% RSLogix 500 project DIGITAL_CONTROL_LOGIC_BAK014.RSS, saved by version 12.00.00.00 %
PROJECT "DRACOFS"    % processor: Bul.1763 MicroLogix 1100 Series B %

PROGRAM FILES
  LAD 2 "MAIN"  3 rungs
  LAD 4 "DIGITAL IO"  5 rungs
  LAD 5 "CONTROL"  10 rungs

DATA FILES
  O0 OUTPUT  5 elements
  I1 INPUT  7 elements
  S2 STATUS  66 elements
  B3 BINARY  1 elements
  T4 TIMER  3 elements
  C5 COUNTER  1 elements
  R6 CONTROL  1 elements
  N7 INTEGER  1 elements
  F8 FLOAT  1 elements

LADDER 2 "MAIN"
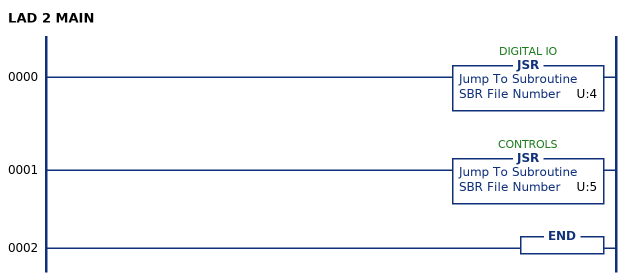
% Rung: 0 %
SOR JSR U:4 EOR
%   U:4  "DIGITAL IO" %
% Rung: 1 %
SOR JSR U:5 EOR
%   U:5  "CONTROLS" %
% Rung: 2 %
SOR END EOR

LADDER 4 "DIGITAL IO"
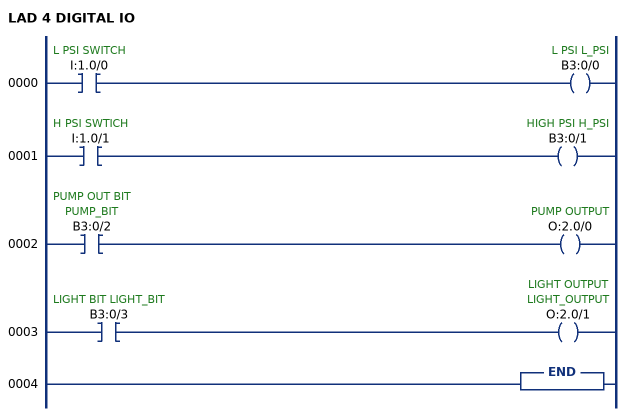
% Rung: 0 %
SOR XIC I:1.0/0 OTE B3:0/0 EOR
%   I:1.0/0  "L PSI SWITCH" %
%   B3:0/0  L_PSI  "L PSI" %
% Rung: 1 %
SOR XIC I:1.0/1 OTE B3:0/1 EOR
%   I:1.0/1  "H PSI SWTICH" %
%   B3:0/1  H_PSI  "HIGH PSI" %
% Rung: 2 %
SOR XIC B3:0/2 OTE O:2.0/0 EOR
%   B3:0/2  PUMP_BIT  "PUMP OUT BIT" %
%   O:2.0/0  "PUMP OUTPUT" %
% Rung: 3 %
SOR XIC B3:0/3 OTE O:2.0/1 EOR
%   B3:0/3  LIGHT_BIT  "LIGHT BIT" %
%   O:2.0/1  LIGHT_OUTPUT  "LIGHT OUTPUT" %
% Rung: 4 %
SOR END EOR

LADDER 5 "CONTROL"
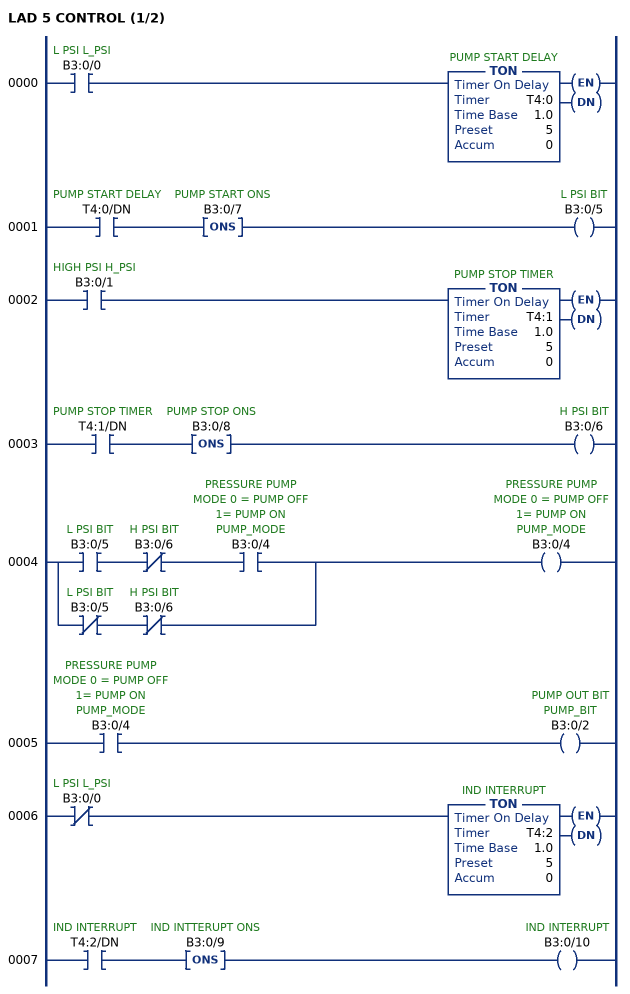
% Rung: 0 %
SOR XIC B3:0/0 TON T4:0 1.0 5 0 EOR
%   B3:0/0  L_PSI  "L PSI" %
%   T4:0  "PUMP START DELAY" %
% Rung: 1 %
SOR XIC T4:0/DN ONS B3:0/7 OTE B3:0/5 EOR
%   T4:0  "PUMP START DELAY" %
%   B3:0/7  "PUMP START ONS" %
%   B3:0/5  "L PSI BIT" %
% Rung: 2 %
SOR XIC B3:0/1 TON T4:1 1.0 5 0 EOR
%   B3:0/1  H_PSI  "HIGH PSI" %
%   T4:1  "PUMP STOP TIMER" %
% Rung: 3 %
SOR XIC T4:1/DN ONS B3:0/8 OTE B3:0/6 EOR
%   T4:1  "PUMP STOP TIMER" %
%   B3:0/8  "PUMP STOP ONS" %
%   B3:0/6  "H PSI BIT" %
% Rung: 4 %
SOR BST XIC B3:0/5 XIO B3:0/6 XIC B3:0/4 NXB XIO B3:0/5 XIO B3:0/6 BND OTE B3:0/4 EOR
%   B3:0/5  "L PSI BIT" %
%   B3:0/6  "H PSI BIT" %
%   B3:0/4  PUMP_MODE  "PRESSURE PUMP MODE 0 = PUMP OFF 1= PUMP ON" %
% Rung: 5 %
SOR XIC B3:0/4 OTE B3:0/2 EOR
%   B3:0/4  PUMP_MODE  "PRESSURE PUMP MODE 0 = PUMP OFF 1= PUMP ON" %
%   B3:0/2  PUMP_BIT  "PUMP OUT BIT" %
% Rung: 6 %
SOR XIO B3:0/0 TON T4:2 1.0 5 0 EOR
%   B3:0/0  L_PSI  "L PSI" %
%   T4:2  "IND INTERRUPT" %
% Rung: 7 %
SOR XIC T4:2/DN ONS B3:0/9 OTE B3:0/10 EOR
%   T4:2  "IND INTERRUPT" %
%   B3:0/9  "IND INTTERUPT ONS" %
%   B3:0/10  "IND INTERRUPT" %

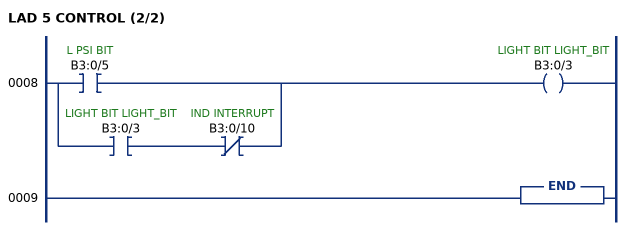
% Rung: 8 %
SOR BST XIC B3:0/5 NXB XIC B3:0/3 XIO B3:0/10 BND OTE B3:0/3 EOR
%   B3:0/5  "L PSI BIT" %
%   B3:0/3  LIGHT_BIT  "LIGHT BIT" %
%   B3:0/10  "IND INTERRUPT" %
% Rung: 9 %
SOR END EOR

DATA TABLE (non-zero values as saved)
DATA B3
% B3:0 % 0X0068
DATA T4
% .PRE .ACC %
% T4:0 % 5 0
% T4:1 % 5 0
% T4:2 % 5 0
